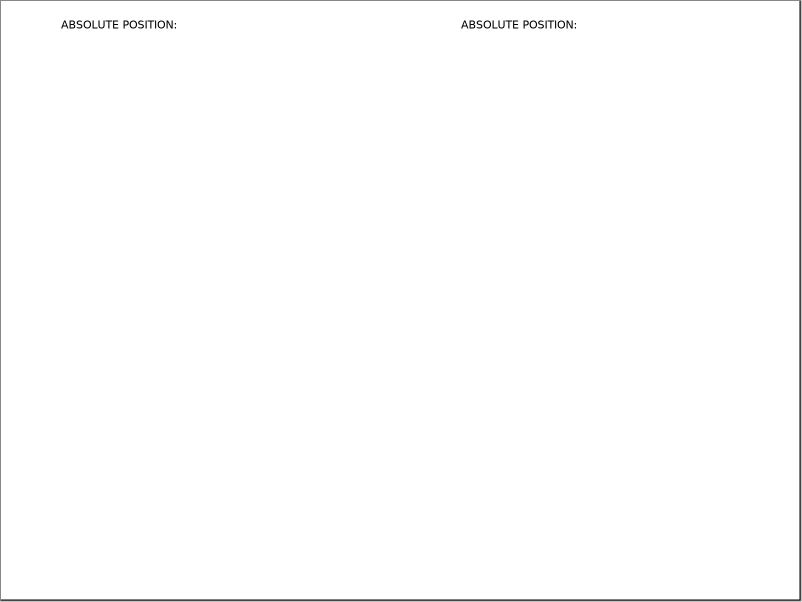
VISUALIZATION F16_Read_Motion_State  // 802x602
    Rectangle (0,0 800x600)
    Label (10,10 170x30), "ABSOLUTE POSITION:"
    Label (410,10 170x30), "ABSOLUTE POSITION:"
END_VISUALIZATION

(* stored: Version 1.1.0.1, ProductVersion 3.1.4022.7
   Visu F16_Read_Motion_State: Id {5cf1740c-3858-4a2e-83fa-1dab314d6ef5} *)
